TYPE ST_FillOrder :
STRUCT
	bActive		: BOOL;
	//dtTimeStamp	: DT;
	//eLevel		: E_LogLevel;
	//sSource		: STRING(31);
	//sMessage 	: T_MaxString;
END_STRUCT
END_TYPE

(* stored: Version 1.1.0.1, ProductVersion 3.1.4024.12
   DUT ST_FillOrder: Id {603e2410-8bf9-4287-a816-3db2ad45c753} *)
